// TIA Portal V17 export
// export: Created 2025-03-07T09:17:59.3981657Z, ExportSetting WithDefaults, DisplayName Totally Integrated Automation Portal, DisplayVersion V17 Update 8, DisplayName TIA Portal Openness, DisplayVersion V17 Update 8, DisplayName TIA Portal Version Control Interface, DisplayVersion V17, DisplayName SINAMICS Startdrive Advanced, DisplayVersion V17 SP2, DisplayName SINAMICS Startdrive G110M, G120, G120C, G120D, G120P, G115D, DisplayVersion V17 SP2, DisplayName SINAMICS Startdrive G130, G150, S120, S150, SINAMICS MV, S210, DisplayVersion V17 SP2, DisplayName STEP 7 Professional, DisplayVersion V17 Update 8, DisplayName SINUMERIK ONE STEP 7 Toolbox, DisplayVersion V17 Update 12, DisplayName SINUMERIK 840D sl STEP 7 Toolbox, DisplayVersion V17 Update 12, DisplayName STEP 7 Safety, DisplayVersion V17 Update 6, DisplayName WinCC Advanced, DisplayVersion V17 Update 8
FUNCTION "FC1222_NOZZLE_CLEAN_CYCLE_UNIT_ 01_CLADDING" : Void   // FC1222, LAD
{ S7_Optimized_Access := 'FALSE' }
AUTHOR : ETXETAR
VERSION : 1.0
// stored: AutoNumber false, IsIECCheckEnabled false, SetENOAutomatically false, UDAEnableTagReadback false
   VAR CONSTANT
      FC_NUMBER : DInt := 1222;
   END_VAR
   VAR_TEMP   // added for the SCL form of the ladder/FBD networks
      _w1 : Bool;
      _w2 : Bool;
      _w3 : Bool;
      _w4 : Bool;
   END_VAR
BEGIN

REGION Network 1: GENERAL CONDITIONS
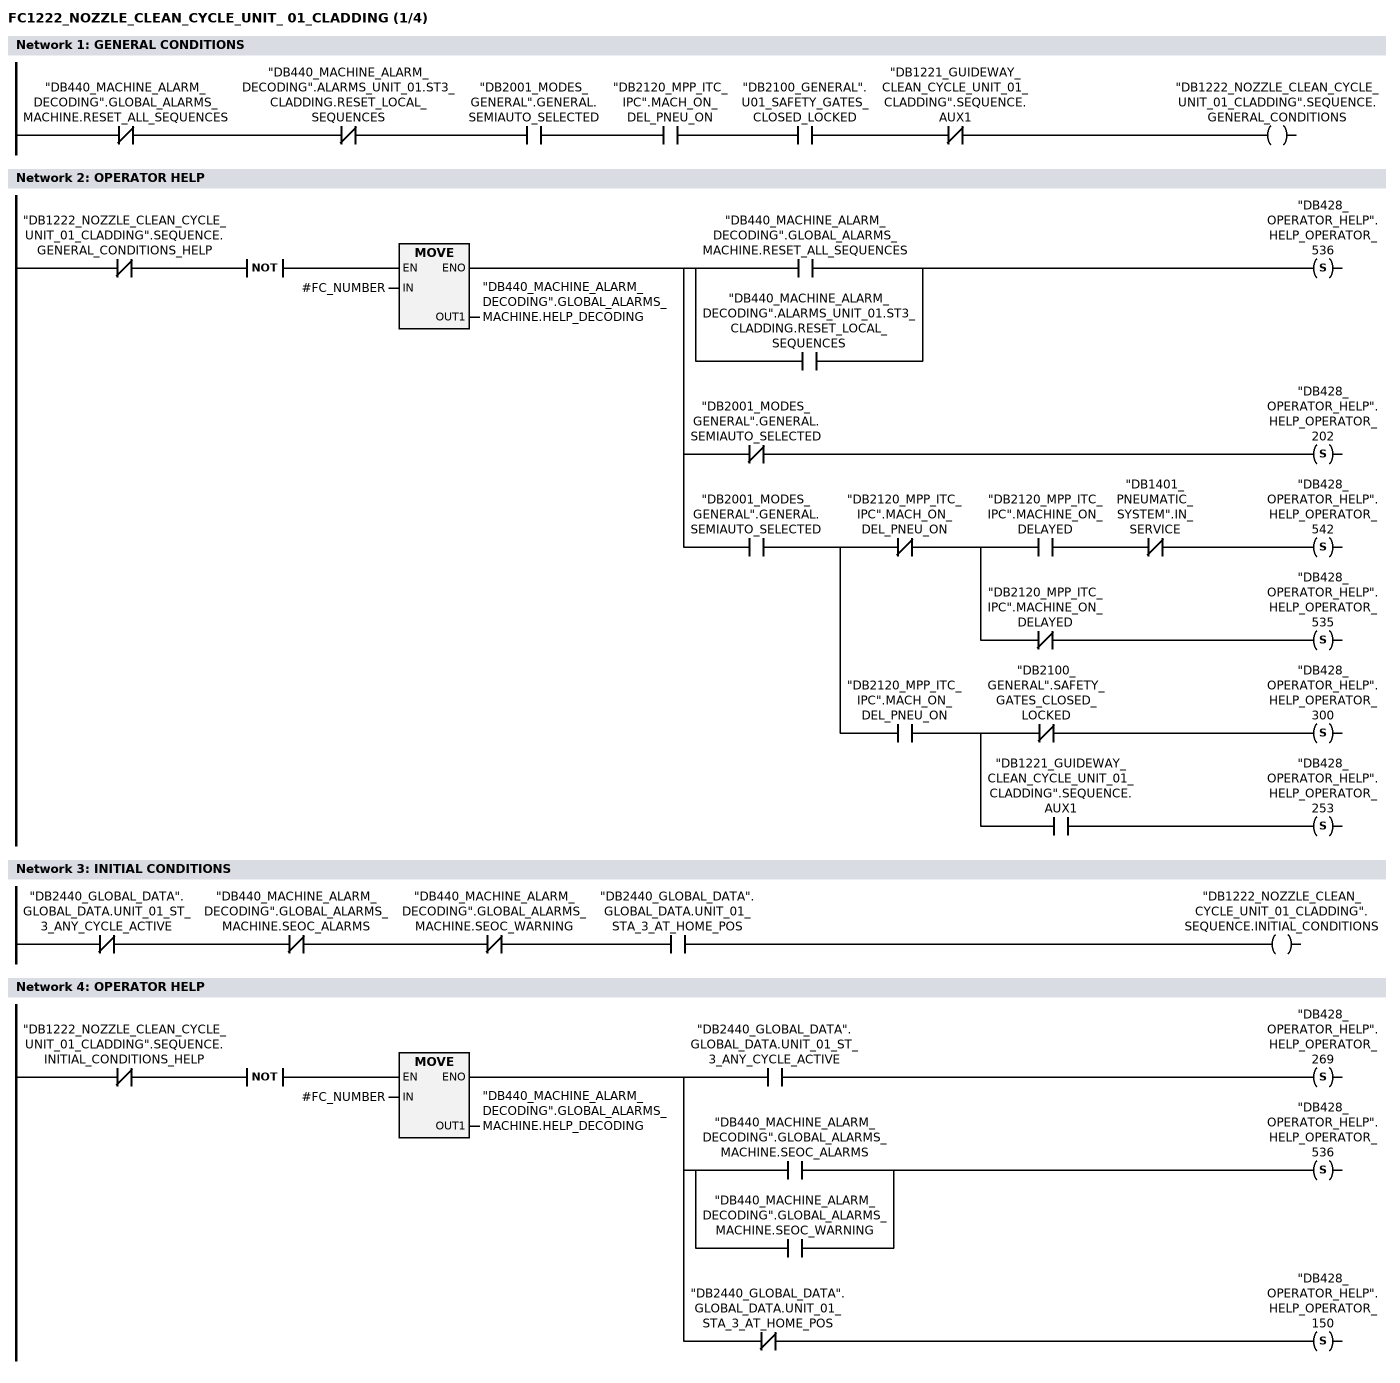
   RUNG wire#powerrail
      I_Contact( "DB440_MACHINE_ALARM_DECODING".GLOBAL_ALARMS_MACHINE.RESET_ALL_SEQUENCES )
      I_Contact( "DB440_MACHINE_ALARM_DECODING".ALARMS_UNIT_01.ST3_CLADDING.RESET_LOCAL_SEQUENCES )
      Contact( "DB2001_MODES_GENERAL".GENERAL.SEMIAUTO_SELECTED )
      Contact( "DB2120_MPP_ITC_IPC".MACH_ON_DEL_PNEU_ON )
      Contact( "DB2100_GENERAL".U01_SAFETY_GATES_CLOSED_LOCKED )
      I_Contact( "DB1221_GUIDEWAY_CLEAN_CYCLE_UNIT_01_CLADDING".SEQUENCE.AUX1 )
      Coil( "DB1222_NOZZLE_CLEAN_CYCLE_UNIT_01_CLADDING".SEQUENCE.GENERAL_CONDITIONS )
   END_RUNG
   // the same network as SCL:
   "DB1222_NOZZLE_CLEAN_CYCLE_UNIT_01_CLADDING".SEQUENCE.GENERAL_CONDITIONS := NOT "DB440_MACHINE_ALARM_DECODING".GLOBAL_ALARMS_MACHINE.RESET_ALL_SEQUENCES AND NOT "DB440_MACHINE_ALARM_DECODING".ALARMS_UNIT_01.ST3_CLADDING.RESET_LOCAL_SEQUENCES AND "DB2001_MODES_GENERAL".GENERAL.SEMIAUTO_SELECTED AND "DB2120_MPP_ITC_IPC".MACH_ON_DEL_PNEU_ON AND "DB2100_GENERAL".U01_SAFETY_GATES_CLOSED_LOCKED AND NOT "DB1221_GUIDEWAY_CLEAN_CYCLE_UNIT_01_CLADDING".SEQUENCE.AUX1;
END_REGION

REGION Network 2: OPERATOR HELP
   RUNG wire#powerrail
      I_Contact( "DB1222_NOZZLE_CLEAN_CYCLE_UNIT_01_CLADDING".SEQUENCE.GENERAL_CONDITIONS_HELP )
      Not()
      { S7_GenerateENO := "TRUE" } Move(in := #FC_NUMBER, out1 => "DB440_MACHINE_ALARM_DECODING".GLOBAL_ALARMS_MACHINE.HELP_DECODING)
      wire#w1
      Contact( "DB440_MACHINE_ALARM_DECODING".GLOBAL_ALARMS_MACHINE.RESET_ALL_SEQUENCES )
      wire#w2
      S_Coil( "DB428_OPERATOR_HELP".HELP_OPERATOR_536 )
   END_RUNG
   RUNG wire#w1
      Contact( "DB440_MACHINE_ALARM_DECODING".ALARMS_UNIT_01.ST3_CLADDING.RESET_LOCAL_SEQUENCES )
   END_RUNG wire#w2
   RUNG wire#w1
      I_Contact( "DB2001_MODES_GENERAL".GENERAL.SEMIAUTO_SELECTED )
      S_Coil( "DB428_OPERATOR_HELP".HELP_OPERATOR_202 )
   END_RUNG
   RUNG wire#w1
      Contact( "DB2001_MODES_GENERAL".GENERAL.SEMIAUTO_SELECTED )
      wire#w3
      I_Contact( "DB2120_MPP_ITC_IPC".MACH_ON_DEL_PNEU_ON )
      wire#w4
      Contact( "DB2120_MPP_ITC_IPC".MACHINE_ON_DELAYED )
      I_Contact( "DB1401_PNEUMATIC_SYSTEM".IN_SERVICE )
      S_Coil( "DB428_OPERATOR_HELP".HELP_OPERATOR_542 )
   END_RUNG
   RUNG wire#w4
      I_Contact( "DB2120_MPP_ITC_IPC".MACHINE_ON_DELAYED )
      S_Coil( "DB428_OPERATOR_HELP".HELP_OPERATOR_535 )
   END_RUNG
   RUNG wire#w3
      Contact( "DB2120_MPP_ITC_IPC".MACH_ON_DEL_PNEU_ON )
      wire#w5
      I_Contact( "DB2100_GENERAL".SAFETY_GATES_CLOSED_LOCKED )
      S_Coil( "DB428_OPERATOR_HELP".HELP_OPERATOR_300 )
   END_RUNG
   RUNG wire#w5
      Contact( "DB1221_GUIDEWAY_CLEAN_CYCLE_UNIT_01_CLADDING".SEQUENCE.AUX1 )
      S_Coil( "DB428_OPERATOR_HELP".HELP_OPERATOR_253 )
   END_RUNG
   // the same network as SCL:
   // ENO of a box is taken as its EN; it also drops when the box reports an error
   #_w1 := NOT (NOT "DB1222_NOZZLE_CLEAN_CYCLE_UNIT_01_CLADDING".SEQUENCE.GENERAL_CONDITIONS_HELP);
   IF #_w1 THEN "DB440_MACHINE_ALARM_DECODING".GLOBAL_ALARMS_MACHINE.HELP_DECODING := #FC_NUMBER; END_IF;
   IF #_w1 AND ("DB440_MACHINE_ALARM_DECODING".GLOBAL_ALARMS_MACHINE.RESET_ALL_SEQUENCES OR "DB440_MACHINE_ALARM_DECODING".ALARMS_UNIT_01.ST3_CLADDING.RESET_LOCAL_SEQUENCES) THEN
       "DB428_OPERATOR_HELP".HELP_OPERATOR_536 := TRUE;
   END_IF;
   IF #_w1 AND NOT "DB2001_MODES_GENERAL".GENERAL.SEMIAUTO_SELECTED THEN
       "DB428_OPERATOR_HELP".HELP_OPERATOR_202 := TRUE;
   END_IF;
   #_w2 := #_w1 AND "DB2001_MODES_GENERAL".GENERAL.SEMIAUTO_SELECTED;
   #_w3 := #_w2 AND NOT "DB2120_MPP_ITC_IPC".MACH_ON_DEL_PNEU_ON;
   IF #_w3 AND "DB2120_MPP_ITC_IPC".MACHINE_ON_DELAYED AND NOT "DB1401_PNEUMATIC_SYSTEM".IN_SERVICE THEN
       "DB428_OPERATOR_HELP".HELP_OPERATOR_542 := TRUE;
   END_IF;
   IF #_w3 AND NOT "DB2120_MPP_ITC_IPC".MACHINE_ON_DELAYED THEN
       "DB428_OPERATOR_HELP".HELP_OPERATOR_535 := TRUE;
   END_IF;
   #_w4 := #_w2 AND "DB2120_MPP_ITC_IPC".MACH_ON_DEL_PNEU_ON;
   IF #_w4 AND NOT "DB2100_GENERAL".SAFETY_GATES_CLOSED_LOCKED THEN
       "DB428_OPERATOR_HELP".HELP_OPERATOR_300 := TRUE;
   END_IF;
   IF #_w4 AND "DB1221_GUIDEWAY_CLEAN_CYCLE_UNIT_01_CLADDING".SEQUENCE.AUX1 THEN
       "DB428_OPERATOR_HELP".HELP_OPERATOR_253 := TRUE;
   END_IF;
END_REGION

REGION Network 3: INITIAL CONDITIONS
   RUNG wire#powerrail
      I_Contact( "DB2440_GLOBAL_DATA".GLOBAL_DATA.UNIT_01_ST_3_ANY_CYCLE_ACTIVE )
      I_Contact( "DB440_MACHINE_ALARM_DECODING".GLOBAL_ALARMS_MACHINE.SEOC_ALARMS )
      I_Contact( "DB440_MACHINE_ALARM_DECODING".GLOBAL_ALARMS_MACHINE.SEOC_WARNING )
      Contact( "DB2440_GLOBAL_DATA".GLOBAL_DATA.UNIT_01_STA_3_AT_HOME_POS )
      Coil( "DB1222_NOZZLE_CLEAN_CYCLE_UNIT_01_CLADDING".SEQUENCE.INITIAL_CONDITIONS )
   END_RUNG
   // the same network as SCL:
   "DB1222_NOZZLE_CLEAN_CYCLE_UNIT_01_CLADDING".SEQUENCE.INITIAL_CONDITIONS := NOT "DB2440_GLOBAL_DATA".GLOBAL_DATA.UNIT_01_ST_3_ANY_CYCLE_ACTIVE AND NOT "DB440_MACHINE_ALARM_DECODING".GLOBAL_ALARMS_MACHINE.SEOC_ALARMS AND NOT "DB440_MACHINE_ALARM_DECODING".GLOBAL_ALARMS_MACHINE.SEOC_WARNING AND "DB2440_GLOBAL_DATA".GLOBAL_DATA.UNIT_01_STA_3_AT_HOME_POS;
END_REGION

REGION Network 4: OPERATOR HELP
   RUNG wire#powerrail
      I_Contact( "DB1222_NOZZLE_CLEAN_CYCLE_UNIT_01_CLADDING".SEQUENCE.INITIAL_CONDITIONS_HELP )
      Not()
      { S7_GenerateENO := "TRUE" } Move(in := #FC_NUMBER, out1 => "DB440_MACHINE_ALARM_DECODING".GLOBAL_ALARMS_MACHINE.HELP_DECODING)
      wire#w1
      Contact( "DB2440_GLOBAL_DATA".GLOBAL_DATA.UNIT_01_ST_3_ANY_CYCLE_ACTIVE )
      S_Coil( "DB428_OPERATOR_HELP".HELP_OPERATOR_269 )
   END_RUNG
   RUNG wire#w1
      Contact( "DB440_MACHINE_ALARM_DECODING".GLOBAL_ALARMS_MACHINE.SEOC_ALARMS )
      wire#w2
      S_Coil( "DB428_OPERATOR_HELP".HELP_OPERATOR_536 )
   END_RUNG
   RUNG wire#w1
      Contact( "DB440_MACHINE_ALARM_DECODING".GLOBAL_ALARMS_MACHINE.SEOC_WARNING )
   END_RUNG wire#w2
   RUNG wire#w1
      I_Contact( "DB2440_GLOBAL_DATA".GLOBAL_DATA.UNIT_01_STA_3_AT_HOME_POS )
      S_Coil( "DB428_OPERATOR_HELP".HELP_OPERATOR_150 )
   END_RUNG
   // the same network as SCL:
   // ENO of a box is taken as its EN; it also drops when the box reports an error
   #_w1 := NOT (NOT "DB1222_NOZZLE_CLEAN_CYCLE_UNIT_01_CLADDING".SEQUENCE.INITIAL_CONDITIONS_HELP);
   IF #_w1 THEN "DB440_MACHINE_ALARM_DECODING".GLOBAL_ALARMS_MACHINE.HELP_DECODING := #FC_NUMBER; END_IF;
   IF #_w1 AND "DB2440_GLOBAL_DATA".GLOBAL_DATA.UNIT_01_ST_3_ANY_CYCLE_ACTIVE THEN
       "DB428_OPERATOR_HELP".HELP_OPERATOR_269 := TRUE;
   END_IF;
   IF #_w1 AND ("DB440_MACHINE_ALARM_DECODING".GLOBAL_ALARMS_MACHINE.SEOC_ALARMS OR "DB440_MACHINE_ALARM_DECODING".GLOBAL_ALARMS_MACHINE.SEOC_WARNING) THEN
       "DB428_OPERATOR_HELP".HELP_OPERATOR_536 := TRUE;
   END_IF;
   IF #_w1 AND NOT "DB2440_GLOBAL_DATA".GLOBAL_DATA.UNIT_01_STA_3_AT_HOME_POS THEN
       "DB428_OPERATOR_HELP".HELP_OPERATOR_150 := TRUE;
   END_IF;
END_REGION

REGION Network 5: SEMI AUTO REQUEST
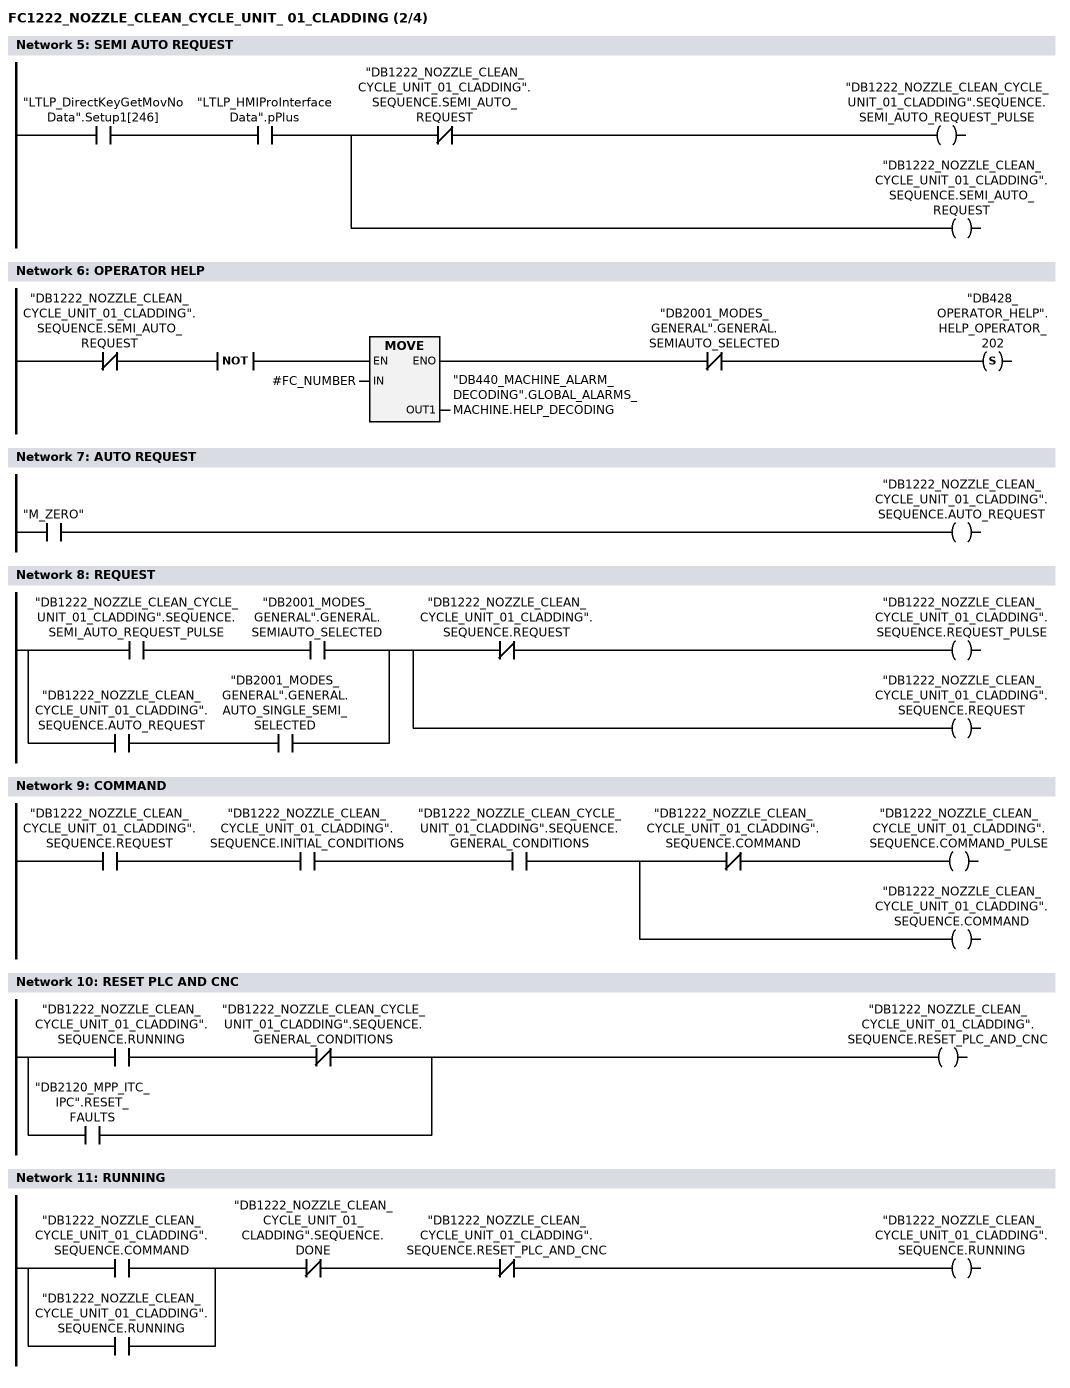
   RUNG wire#powerrail
      Contact( "LTLP_DirectKeyGetMovNoData".Setup1[246] )
      Contact( "LTLP_HMIProInterfaceData".pPlus )
      wire#w1
      I_Contact( "DB1222_NOZZLE_CLEAN_CYCLE_UNIT_01_CLADDING".SEQUENCE.SEMI_AUTO_REQUEST )
      Coil( "DB1222_NOZZLE_CLEAN_CYCLE_UNIT_01_CLADDING".SEQUENCE.SEMI_AUTO_REQUEST_PULSE )
   END_RUNG
   RUNG wire#w1
      Coil( "DB1222_NOZZLE_CLEAN_CYCLE_UNIT_01_CLADDING".SEQUENCE.SEMI_AUTO_REQUEST )
   END_RUNG
   // the same network as SCL:
   #_w1 := "LTLP_DirectKeyGetMovNoData".Setup1[246] AND "LTLP_HMIProInterfaceData".pPlus;
   "DB1222_NOZZLE_CLEAN_CYCLE_UNIT_01_CLADDING".SEQUENCE.SEMI_AUTO_REQUEST_PULSE := #_w1 AND NOT "DB1222_NOZZLE_CLEAN_CYCLE_UNIT_01_CLADDING".SEQUENCE.SEMI_AUTO_REQUEST;
   "DB1222_NOZZLE_CLEAN_CYCLE_UNIT_01_CLADDING".SEQUENCE.SEMI_AUTO_REQUEST := #_w1;
END_REGION

REGION Network 6: OPERATOR HELP
   RUNG wire#powerrail
      I_Contact( "DB1222_NOZZLE_CLEAN_CYCLE_UNIT_01_CLADDING".SEQUENCE.SEMI_AUTO_REQUEST )
      Not()
      { S7_GenerateENO := "TRUE" } Move(in := #FC_NUMBER, out1 => "DB440_MACHINE_ALARM_DECODING".GLOBAL_ALARMS_MACHINE.HELP_DECODING)
      I_Contact( "DB2001_MODES_GENERAL".GENERAL.SEMIAUTO_SELECTED )
      S_Coil( "DB428_OPERATOR_HELP".HELP_OPERATOR_202 )
   END_RUNG
   // the same network as SCL:
   // ENO of a box is taken as its EN; it also drops when the box reports an error
   #_w1 := NOT (NOT "DB1222_NOZZLE_CLEAN_CYCLE_UNIT_01_CLADDING".SEQUENCE.SEMI_AUTO_REQUEST);
   IF #_w1 THEN "DB440_MACHINE_ALARM_DECODING".GLOBAL_ALARMS_MACHINE.HELP_DECODING := #FC_NUMBER; END_IF;
   IF #_w1 AND NOT "DB2001_MODES_GENERAL".GENERAL.SEMIAUTO_SELECTED THEN
       "DB428_OPERATOR_HELP".HELP_OPERATOR_202 := TRUE;
   END_IF;
END_REGION

REGION Network 7: AUTO REQUEST
   RUNG wire#powerrail
      Contact( "M_ZERO" )
      Coil( "DB1222_NOZZLE_CLEAN_CYCLE_UNIT_01_CLADDING".SEQUENCE.AUTO_REQUEST )
   END_RUNG
   // the same network as SCL:
   "DB1222_NOZZLE_CLEAN_CYCLE_UNIT_01_CLADDING".SEQUENCE.AUTO_REQUEST := "M_ZERO";
END_REGION

REGION Network 8: REQUEST
   RUNG wire#powerrail
      Contact( "DB1222_NOZZLE_CLEAN_CYCLE_UNIT_01_CLADDING".SEQUENCE.SEMI_AUTO_REQUEST_PULSE )
      Contact( "DB2001_MODES_GENERAL".GENERAL.SEMIAUTO_SELECTED )
      wire#w1
      I_Contact( "DB1222_NOZZLE_CLEAN_CYCLE_UNIT_01_CLADDING".SEQUENCE.REQUEST )
      Coil( "DB1222_NOZZLE_CLEAN_CYCLE_UNIT_01_CLADDING".SEQUENCE.REQUEST_PULSE )
   END_RUNG
   RUNG wire#powerrail
      Contact( "DB1222_NOZZLE_CLEAN_CYCLE_UNIT_01_CLADDING".SEQUENCE.AUTO_REQUEST )
      Contact( "DB2001_MODES_GENERAL".GENERAL.AUTO_SINGLE_SEMI_SELECTED )
   END_RUNG wire#w1
   RUNG wire#w1
      Coil( "DB1222_NOZZLE_CLEAN_CYCLE_UNIT_01_CLADDING".SEQUENCE.REQUEST )
   END_RUNG
   // the same network as SCL:
   #_w1 := ("DB1222_NOZZLE_CLEAN_CYCLE_UNIT_01_CLADDING".SEQUENCE.SEMI_AUTO_REQUEST_PULSE AND "DB2001_MODES_GENERAL".GENERAL.SEMIAUTO_SELECTED) OR ("DB1222_NOZZLE_CLEAN_CYCLE_UNIT_01_CLADDING".SEQUENCE.AUTO_REQUEST AND "DB2001_MODES_GENERAL".GENERAL.AUTO_SINGLE_SEMI_SELECTED);
   "DB1222_NOZZLE_CLEAN_CYCLE_UNIT_01_CLADDING".SEQUENCE.REQUEST_PULSE := #_w1 AND NOT "DB1222_NOZZLE_CLEAN_CYCLE_UNIT_01_CLADDING".SEQUENCE.REQUEST;
   "DB1222_NOZZLE_CLEAN_CYCLE_UNIT_01_CLADDING".SEQUENCE.REQUEST := #_w1;
END_REGION

REGION Network 9: COMMAND
   RUNG wire#powerrail
      Contact( "DB1222_NOZZLE_CLEAN_CYCLE_UNIT_01_CLADDING".SEQUENCE.REQUEST )
      Contact( "DB1222_NOZZLE_CLEAN_CYCLE_UNIT_01_CLADDING".SEQUENCE.INITIAL_CONDITIONS )
      Contact( "DB1222_NOZZLE_CLEAN_CYCLE_UNIT_01_CLADDING".SEQUENCE.GENERAL_CONDITIONS )
      wire#w1
      I_Contact( "DB1222_NOZZLE_CLEAN_CYCLE_UNIT_01_CLADDING".SEQUENCE.COMMAND )
      Coil( "DB1222_NOZZLE_CLEAN_CYCLE_UNIT_01_CLADDING".SEQUENCE.COMMAND_PULSE )
   END_RUNG
   RUNG wire#w1
      Coil( "DB1222_NOZZLE_CLEAN_CYCLE_UNIT_01_CLADDING".SEQUENCE.COMMAND )
   END_RUNG
   // the same network as SCL:
   #_w1 := "DB1222_NOZZLE_CLEAN_CYCLE_UNIT_01_CLADDING".SEQUENCE.REQUEST AND "DB1222_NOZZLE_CLEAN_CYCLE_UNIT_01_CLADDING".SEQUENCE.INITIAL_CONDITIONS AND "DB1222_NOZZLE_CLEAN_CYCLE_UNIT_01_CLADDING".SEQUENCE.GENERAL_CONDITIONS;
   "DB1222_NOZZLE_CLEAN_CYCLE_UNIT_01_CLADDING".SEQUENCE.COMMAND_PULSE := #_w1 AND NOT "DB1222_NOZZLE_CLEAN_CYCLE_UNIT_01_CLADDING".SEQUENCE.COMMAND;
   "DB1222_NOZZLE_CLEAN_CYCLE_UNIT_01_CLADDING".SEQUENCE.COMMAND := #_w1;
END_REGION

REGION Network 10: RESET PLC AND CNC
   RUNG wire#powerrail
      Contact( "DB1222_NOZZLE_CLEAN_CYCLE_UNIT_01_CLADDING".SEQUENCE.RUNNING )
      I_Contact( "DB1222_NOZZLE_CLEAN_CYCLE_UNIT_01_CLADDING".SEQUENCE.GENERAL_CONDITIONS )
      wire#w1
      Coil( "DB1222_NOZZLE_CLEAN_CYCLE_UNIT_01_CLADDING".SEQUENCE.RESET_PLC_AND_CNC )
   END_RUNG
   RUNG wire#powerrail
      Contact( "DB2120_MPP_ITC_IPC".RESET_FAULTS )
   END_RUNG wire#w1
   // the same network as SCL:
   "DB1222_NOZZLE_CLEAN_CYCLE_UNIT_01_CLADDING".SEQUENCE.RESET_PLC_AND_CNC := ("DB1222_NOZZLE_CLEAN_CYCLE_UNIT_01_CLADDING".SEQUENCE.RUNNING AND NOT "DB1222_NOZZLE_CLEAN_CYCLE_UNIT_01_CLADDING".SEQUENCE.GENERAL_CONDITIONS) OR "DB2120_MPP_ITC_IPC".RESET_FAULTS;
END_REGION

REGION Network 11: RUNNING
   RUNG wire#powerrail
      Contact( "DB1222_NOZZLE_CLEAN_CYCLE_UNIT_01_CLADDING".SEQUENCE.COMMAND )
      wire#w1
      I_Contact( "DB1222_NOZZLE_CLEAN_CYCLE_UNIT_01_CLADDING".SEQUENCE.DONE )
      I_Contact( "DB1222_NOZZLE_CLEAN_CYCLE_UNIT_01_CLADDING".SEQUENCE.RESET_PLC_AND_CNC )
      Coil( "DB1222_NOZZLE_CLEAN_CYCLE_UNIT_01_CLADDING".SEQUENCE.RUNNING )
   END_RUNG
   RUNG wire#powerrail
      Contact( "DB1222_NOZZLE_CLEAN_CYCLE_UNIT_01_CLADDING".SEQUENCE.RUNNING )
   END_RUNG wire#w1
   // the same network as SCL:
   "DB1222_NOZZLE_CLEAN_CYCLE_UNIT_01_CLADDING".SEQUENCE.RUNNING := ("DB1222_NOZZLE_CLEAN_CYCLE_UNIT_01_CLADDING".SEQUENCE.COMMAND OR "DB1222_NOZZLE_CLEAN_CYCLE_UNIT_01_CLADDING".SEQUENCE.RUNNING) AND NOT "DB1222_NOZZLE_CLEAN_CYCLE_UNIT_01_CLADDING".SEQUENCE.DONE AND NOT "DB1222_NOZZLE_CLEAN_CYCLE_UNIT_01_CLADDING".SEQUENCE.RESET_PLC_AND_CNC;
END_REGION

REGION Network 12: STEP 1 SELECT PROGRAM
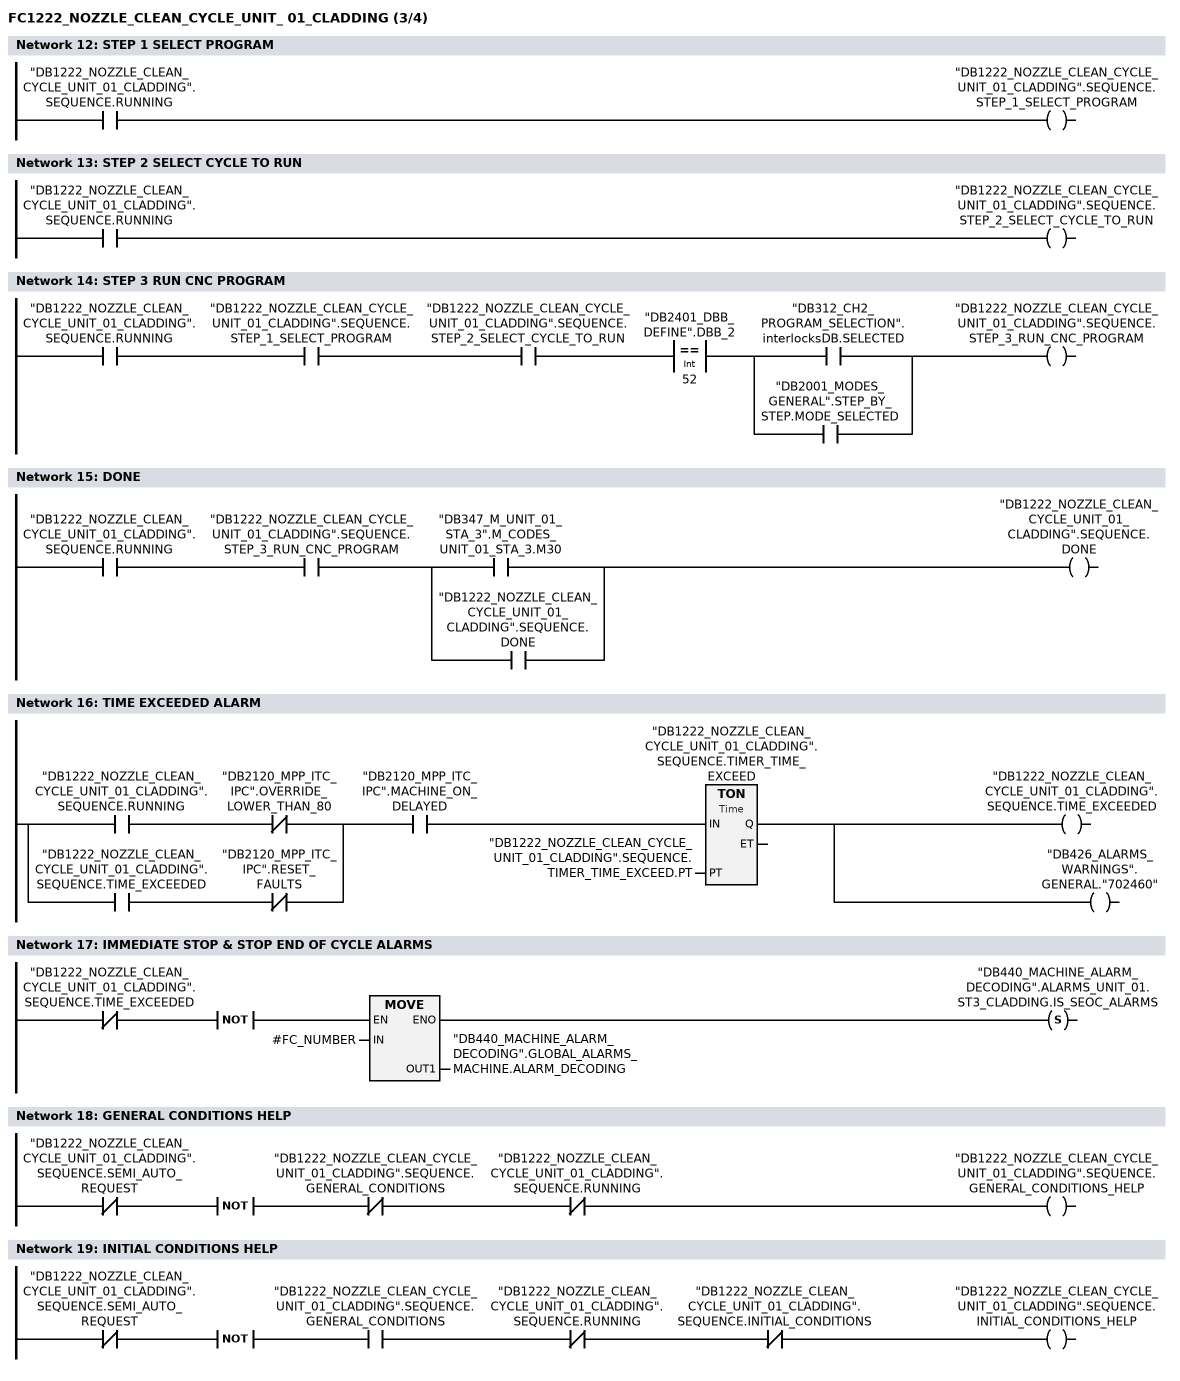
   RUNG wire#powerrail
      Contact( "DB1222_NOZZLE_CLEAN_CYCLE_UNIT_01_CLADDING".SEQUENCE.RUNNING )
      Coil( "DB1222_NOZZLE_CLEAN_CYCLE_UNIT_01_CLADDING".SEQUENCE.STEP_1_SELECT_PROGRAM )
   END_RUNG
   // the same network as SCL:
   "DB1222_NOZZLE_CLEAN_CYCLE_UNIT_01_CLADDING".SEQUENCE.STEP_1_SELECT_PROGRAM := "DB1222_NOZZLE_CLEAN_CYCLE_UNIT_01_CLADDING".SEQUENCE.RUNNING;
END_REGION

REGION Network 13: STEP 2 SELECT CYCLE TO RUN
   RUNG wire#powerrail
      Contact( "DB1222_NOZZLE_CLEAN_CYCLE_UNIT_01_CLADDING".SEQUENCE.RUNNING )
      Coil( "DB1222_NOZZLE_CLEAN_CYCLE_UNIT_01_CLADDING".SEQUENCE.STEP_2_SELECT_CYCLE_TO_RUN )
   END_RUNG
   // the same network as SCL:
   "DB1222_NOZZLE_CLEAN_CYCLE_UNIT_01_CLADDING".SEQUENCE.STEP_2_SELECT_CYCLE_TO_RUN := "DB1222_NOZZLE_CLEAN_CYCLE_UNIT_01_CLADDING".SEQUENCE.RUNNING;
END_REGION

REGION Network 14: STEP 3 RUN CNC PROGRAM
   RUNG wire#powerrail
      Contact( "DB1222_NOZZLE_CLEAN_CYCLE_UNIT_01_CLADDING".SEQUENCE.RUNNING )
      Contact( "DB1222_NOZZLE_CLEAN_CYCLE_UNIT_01_CLADDING".SEQUENCE.STEP_1_SELECT_PROGRAM )
      Contact( "DB1222_NOZZLE_CLEAN_CYCLE_UNIT_01_CLADDING".SEQUENCE.STEP_2_SELECT_CYCLE_TO_RUN )
      { S7_Templates := "SrcType := Int" } EQ_Contact(in1 := "DB2401_DBB_DEFINE".DBB_2, in2 := 52)
      wire#w1
      Contact( "DB312_CH2_PROGRAM_SELECTION".interlocksDB.SELECTED )
      wire#w2
      Coil( "DB1222_NOZZLE_CLEAN_CYCLE_UNIT_01_CLADDING".SEQUENCE.STEP_3_RUN_CNC_PROGRAM )
   END_RUNG
   RUNG wire#w1
      Contact( "DB2001_MODES_GENERAL".STEP_BY_STEP.MODE_SELECTED )
   END_RUNG wire#w2
   // the same network as SCL:
   "DB1222_NOZZLE_CLEAN_CYCLE_UNIT_01_CLADDING".SEQUENCE.STEP_3_RUN_CNC_PROGRAM := "DB1222_NOZZLE_CLEAN_CYCLE_UNIT_01_CLADDING".SEQUENCE.RUNNING AND "DB1222_NOZZLE_CLEAN_CYCLE_UNIT_01_CLADDING".SEQUENCE.STEP_1_SELECT_PROGRAM AND "DB1222_NOZZLE_CLEAN_CYCLE_UNIT_01_CLADDING".SEQUENCE.STEP_2_SELECT_CYCLE_TO_RUN AND ("DB2401_DBB_DEFINE".DBB_2 = 52) AND ("DB312_CH2_PROGRAM_SELECTION".interlocksDB.SELECTED OR "DB2001_MODES_GENERAL".STEP_BY_STEP.MODE_SELECTED);
END_REGION

REGION Network 15: DONE
   RUNG wire#powerrail
      Contact( "DB1222_NOZZLE_CLEAN_CYCLE_UNIT_01_CLADDING".SEQUENCE.RUNNING )
      Contact( "DB1222_NOZZLE_CLEAN_CYCLE_UNIT_01_CLADDING".SEQUENCE.STEP_3_RUN_CNC_PROGRAM )
      wire#w1
      Contact( "DB347_M_UNIT_01_STA_3".M_CODES_UNIT_01_STA_3.M30 )
      wire#w2
      Coil( "DB1222_NOZZLE_CLEAN_CYCLE_UNIT_01_CLADDING".SEQUENCE.DONE )
   END_RUNG
   RUNG wire#w1
      Contact( "DB1222_NOZZLE_CLEAN_CYCLE_UNIT_01_CLADDING".SEQUENCE.DONE )
   END_RUNG wire#w2
   // the same network as SCL:
   "DB1222_NOZZLE_CLEAN_CYCLE_UNIT_01_CLADDING".SEQUENCE.DONE := "DB1222_NOZZLE_CLEAN_CYCLE_UNIT_01_CLADDING".SEQUENCE.RUNNING AND "DB1222_NOZZLE_CLEAN_CYCLE_UNIT_01_CLADDING".SEQUENCE.STEP_3_RUN_CNC_PROGRAM AND ("DB347_M_UNIT_01_STA_3".M_CODES_UNIT_01_STA_3.M30 OR "DB1222_NOZZLE_CLEAN_CYCLE_UNIT_01_CLADDING".SEQUENCE.DONE);
END_REGION

REGION Network 16: TIME EXCEEDED ALARM
   RUNG wire#powerrail
      Contact( "DB1222_NOZZLE_CLEAN_CYCLE_UNIT_01_CLADDING".SEQUENCE.RUNNING )
      I_Contact( "DB2120_MPP_ITC_IPC".OVERRIDE_LOWER_THAN_80 )
      wire#w1
      Contact( "DB2120_MPP_ITC_IPC".MACHINE_ON_DELAYED )
      { S7_Templates := "time_type := Time" } "DB1222_NOZZLE_CLEAN_CYCLE_UNIT_01_CLADDING".SEQUENCE.TIMER_TIME_EXCEED.TON(pt := "DB1222_NOZZLE_CLEAN_CYCLE_UNIT_01_CLADDING".SEQUENCE.TIMER_TIME_EXCEED.PT, et =>)
      wire#w2
      Coil( "DB1222_NOZZLE_CLEAN_CYCLE_UNIT_01_CLADDING".SEQUENCE.TIME_EXCEEDED )
   END_RUNG
   RUNG wire#powerrail
      Contact( "DB1222_NOZZLE_CLEAN_CYCLE_UNIT_01_CLADDING".SEQUENCE.TIME_EXCEEDED )
      I_Contact( "DB2120_MPP_ITC_IPC".RESET_FAULTS )
   END_RUNG wire#w1
   RUNG wire#w2
      Coil( "DB426_ALARMS_WARNINGS".GENERAL."702460" )
   END_RUNG
   // the same network as SCL:
   "DB1222_NOZZLE_CLEAN_CYCLE_UNIT_01_CLADDING".SEQUENCE.TIMER_TIME_EXCEED.TON(IN := (("DB1222_NOZZLE_CLEAN_CYCLE_UNIT_01_CLADDING".SEQUENCE.RUNNING AND NOT "DB2120_MPP_ITC_IPC".OVERRIDE_LOWER_THAN_80) OR ("DB1222_NOZZLE_CLEAN_CYCLE_UNIT_01_CLADDING".SEQUENCE.TIME_EXCEEDED AND NOT "DB2120_MPP_ITC_IPC".RESET_FAULTS)) AND "DB2120_MPP_ITC_IPC".MACHINE_ON_DELAYED,
                           PT := "DB1222_NOZZLE_CLEAN_CYCLE_UNIT_01_CLADDING".SEQUENCE.TIMER_TIME_EXCEED.PT);
   "DB1222_NOZZLE_CLEAN_CYCLE_UNIT_01_CLADDING".SEQUENCE.TIME_EXCEEDED := "DB1222_NOZZLE_CLEAN_CYCLE_UNIT_01_CLADDING".SEQUENCE.TIMER_TIME_EXCEED.Q;
   "DB426_ALARMS_WARNINGS".GENERAL."702460" := "DB1222_NOZZLE_CLEAN_CYCLE_UNIT_01_CLADDING".SEQUENCE.TIMER_TIME_EXCEED.Q;
END_REGION

REGION Network 17: IMMEDIATE STOP & STOP END OF CYCLE ALARMS
   RUNG wire#powerrail
      I_Contact( "DB1222_NOZZLE_CLEAN_CYCLE_UNIT_01_CLADDING".SEQUENCE.TIME_EXCEEDED )
      Not()
      { S7_GenerateENO := "TRUE" } Move(in := #FC_NUMBER, out1 => "DB440_MACHINE_ALARM_DECODING".GLOBAL_ALARMS_MACHINE.ALARM_DECODING)
      S_Coil( "DB440_MACHINE_ALARM_DECODING".ALARMS_UNIT_01.ST3_CLADDING.IS_SEOC_ALARMS )
   END_RUNG
   // the same network as SCL:
   // ENO of a box is taken as its EN; it also drops when the box reports an error
   IF NOT (NOT "DB1222_NOZZLE_CLEAN_CYCLE_UNIT_01_CLADDING".SEQUENCE.TIME_EXCEEDED) THEN
       "DB440_MACHINE_ALARM_DECODING".GLOBAL_ALARMS_MACHINE.ALARM_DECODING := #FC_NUMBER;
       "DB440_MACHINE_ALARM_DECODING".ALARMS_UNIT_01.ST3_CLADDING.IS_SEOC_ALARMS := TRUE;
   END_IF;
END_REGION

REGION Network 18: GENERAL CONDITIONS HELP
   RUNG wire#powerrail
      I_Contact( "DB1222_NOZZLE_CLEAN_CYCLE_UNIT_01_CLADDING".SEQUENCE.SEMI_AUTO_REQUEST )
      Not()
      I_Contact( "DB1222_NOZZLE_CLEAN_CYCLE_UNIT_01_CLADDING".SEQUENCE.GENERAL_CONDITIONS )
      I_Contact( "DB1222_NOZZLE_CLEAN_CYCLE_UNIT_01_CLADDING".SEQUENCE.RUNNING )
      Coil( "DB1222_NOZZLE_CLEAN_CYCLE_UNIT_01_CLADDING".SEQUENCE.GENERAL_CONDITIONS_HELP )
   END_RUNG
   // the same network as SCL:
   "DB1222_NOZZLE_CLEAN_CYCLE_UNIT_01_CLADDING".SEQUENCE.GENERAL_CONDITIONS_HELP := NOT (NOT "DB1222_NOZZLE_CLEAN_CYCLE_UNIT_01_CLADDING".SEQUENCE.SEMI_AUTO_REQUEST) AND NOT "DB1222_NOZZLE_CLEAN_CYCLE_UNIT_01_CLADDING".SEQUENCE.GENERAL_CONDITIONS AND NOT "DB1222_NOZZLE_CLEAN_CYCLE_UNIT_01_CLADDING".SEQUENCE.RUNNING;
END_REGION

REGION Network 19: INITIAL CONDITIONS HELP
   RUNG wire#powerrail
      I_Contact( "DB1222_NOZZLE_CLEAN_CYCLE_UNIT_01_CLADDING".SEQUENCE.SEMI_AUTO_REQUEST )
      Not()
      Contact( "DB1222_NOZZLE_CLEAN_CYCLE_UNIT_01_CLADDING".SEQUENCE.GENERAL_CONDITIONS )
      I_Contact( "DB1222_NOZZLE_CLEAN_CYCLE_UNIT_01_CLADDING".SEQUENCE.RUNNING )
      I_Contact( "DB1222_NOZZLE_CLEAN_CYCLE_UNIT_01_CLADDING".SEQUENCE.INITIAL_CONDITIONS )
      Coil( "DB1222_NOZZLE_CLEAN_CYCLE_UNIT_01_CLADDING".SEQUENCE.INITIAL_CONDITIONS_HELP )
   END_RUNG
   // the same network as SCL:
   "DB1222_NOZZLE_CLEAN_CYCLE_UNIT_01_CLADDING".SEQUENCE.INITIAL_CONDITIONS_HELP := NOT (NOT "DB1222_NOZZLE_CLEAN_CYCLE_UNIT_01_CLADDING".SEQUENCE.SEMI_AUTO_REQUEST) AND "DB1222_NOZZLE_CLEAN_CYCLE_UNIT_01_CLADDING".SEQUENCE.GENERAL_CONDITIONS AND NOT "DB1222_NOZZLE_CLEAN_CYCLE_UNIT_01_CLADDING".SEQUENCE.RUNNING AND NOT "DB1222_NOZZLE_CLEAN_CYCLE_UNIT_01_CLADDING".SEQUENCE.INITIAL_CONDITIONS;
END_REGION

REGION Network 20: HMI STATUS
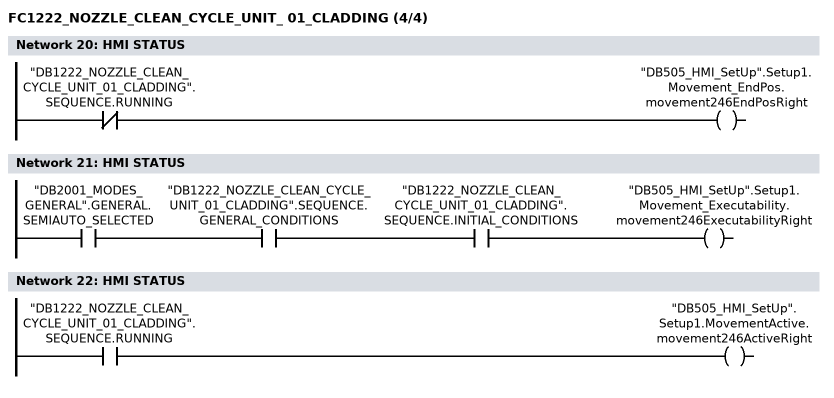
   RUNG wire#powerrail
      I_Contact( "DB1222_NOZZLE_CLEAN_CYCLE_UNIT_01_CLADDING".SEQUENCE.RUNNING )
      Coil( "DB505_HMI_SetUp".Setup1.Movement_EndPos.movement246EndPosRight )
   END_RUNG
   // the same network as SCL:
   "DB505_HMI_SetUp".Setup1.Movement_EndPos.movement246EndPosRight := NOT "DB1222_NOZZLE_CLEAN_CYCLE_UNIT_01_CLADDING".SEQUENCE.RUNNING;
END_REGION

REGION Network 21: HMI STATUS
   RUNG wire#powerrail
      Contact( "DB2001_MODES_GENERAL".GENERAL.SEMIAUTO_SELECTED )
      Contact( "DB1222_NOZZLE_CLEAN_CYCLE_UNIT_01_CLADDING".SEQUENCE.GENERAL_CONDITIONS )
      Contact( "DB1222_NOZZLE_CLEAN_CYCLE_UNIT_01_CLADDING".SEQUENCE.INITIAL_CONDITIONS )
      Coil( "DB505_HMI_SetUp".Setup1.Movement_Executability.movement246ExecutabilityRight )
   END_RUNG
   // the same network as SCL:
   "DB505_HMI_SetUp".Setup1.Movement_Executability.movement246ExecutabilityRight := "DB2001_MODES_GENERAL".GENERAL.SEMIAUTO_SELECTED AND "DB1222_NOZZLE_CLEAN_CYCLE_UNIT_01_CLADDING".SEQUENCE.GENERAL_CONDITIONS AND "DB1222_NOZZLE_CLEAN_CYCLE_UNIT_01_CLADDING".SEQUENCE.INITIAL_CONDITIONS;
END_REGION

REGION Network 22: HMI STATUS
   RUNG wire#powerrail
      Contact( "DB1222_NOZZLE_CLEAN_CYCLE_UNIT_01_CLADDING".SEQUENCE.RUNNING )
      Coil( "DB505_HMI_SetUp".Setup1.MovementActive.movement246ActiveRight )
   END_RUNG
   // the same network as SCL:
   "DB505_HMI_SetUp".Setup1.MovementActive.movement246ActiveRight := "DB1222_NOZZLE_CLEAN_CYCLE_UNIT_01_CLADDING".SEQUENCE.RUNNING;
END_REGION
END_FUNCTION
